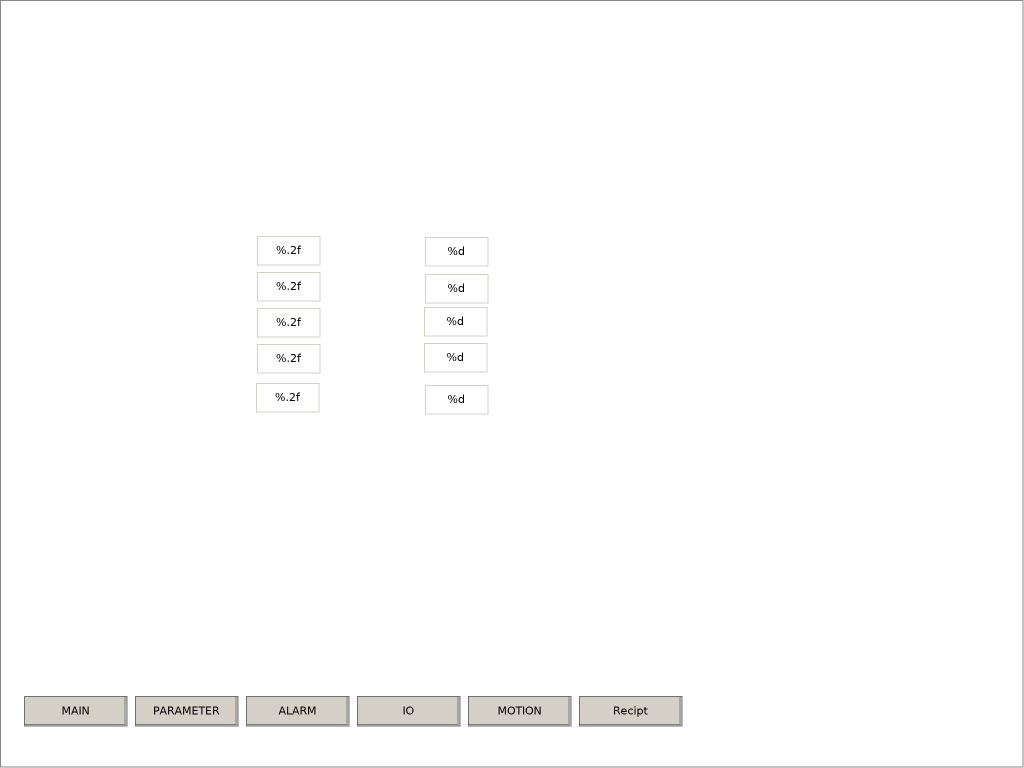
VISUALIZATION PARAMETER  // 1024x768, background image ImagePool_Base.PARAMETER
    Textfield (425,237 63x29), "%d", text variable: MAIN.MFC_delay_show
        OnMouseClick: write the text variable via Default
    Textfield (425,274 63x29), "%d", text variable: MAIN.water_temp_delay_show
        OnMouseClick: write the text variable via Default
    Textfield (424,343 63x29), "%d", text variable: MAIN.WP_delta_delay_show
        OnMouseClick: write the text variable via Default
    Textfield (425,385 63x29), "%d", text variable: MAIN.Heater_temp_delay_show
        OnMouseClick: write the text variable via Default
    Textfield (257,236 63x29), "%.2f", text variable: MAIN.MFC_alarm_setting
        OnMouseClick: write the text variable via Default
    Textfield (257,272 63x29), "%.2f", text variable: MAIN.water_temp_setting
        OnMouseClick: write the text variable via Default
    Textfield (257,308 63x29), "%.2f", text variable: MAIN.WP_delta_setting
        OnMouseClick: write the text variable via Default
    Textfield (257,344 63x29), "%.2f", text variable: MAIN.WP_delta_setting
        OnMouseClick: write the text variable via Default
    Textfield (256,383 63x29), "%.2f", text variable: MAIN.Heater_temp_seeting
        OnMouseClick: write the text variable via Default
    Textfield (424,307 63x29), "%d", text variable: MAIN.WP_delta_delay_show
        OnMouseClick: write the text variable via Default
    Button (24,696 103x30), "MAIN"
        OnMouseClick: change screen: MainBase
    Button (135,696 103x30), "PARAMETER"
        OnMouseClick: change screen: PARAMETER
    Button (246,696 103x30), "ALARM"
        OnMouseClick: change screen: ALARM
    Button (357,696 103x30), "IO"
        OnMouseClick: change screen: IO_TABLE
    Button (468,696 103x30), "MOTION"
        OnMouseClick: change screen: MOTION
    Button (579,696 103x30), "Recipt"
        OnMouseClick: change screen: Recipt
END_VISUALIZATION

(* stored: Version 1.1.0.1, ProductVersion 3.1.4024.12
   Visu PARAMETER: Id {f80e5696-b419-4607-a9fd-1d53b422fd61} *)
